// Mitsubishi GX Works2 project: 워드or   PLC: Q02/Q02H

PROGRAM MAIN
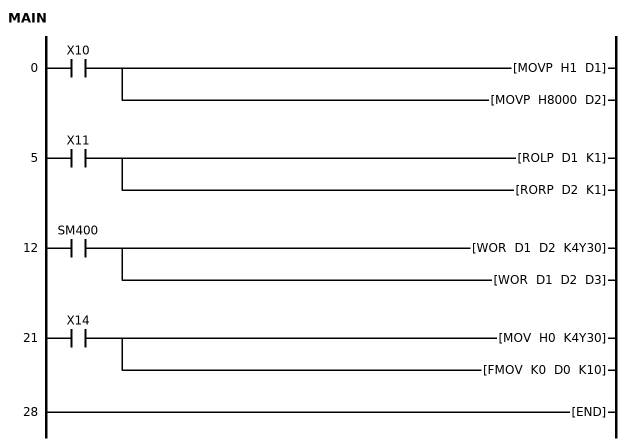
0     LD      X10
      MOVP    H1 D1
      MOVP    H8000 D2
5     LD      X11
      ROLP    D1 K1
      RORP    D2 K1
12    LD      SM400
      WOR     D1 D2 K4Y30
      WOR     D1 D2 D3
21    LD      X14
      MOV     H0 K4Y30
      FMOV    K0 D0 K10
28    END
END_PROGRAM
